PROGRAM MAIN
VAR
END_VAR

END_PROGRAM

(* stored: Version 1.1.0.1
   POU MAIN: Id {3aaccdf2-8248-4196-882d-83f4a667167f} *)
